Staubli VAL3: onStart.pgx

program onStart()
begin
  call language2:setLanguage(language2:libPath()+"/"+saveData:language)
  if save:nBoxType<1 or save:nBoxType>2
    save:nBoxType=1
  endIf
  // reset the Key pressure
  call use:nullKey(nKey)
  //bulidList
  call buildList()
end
